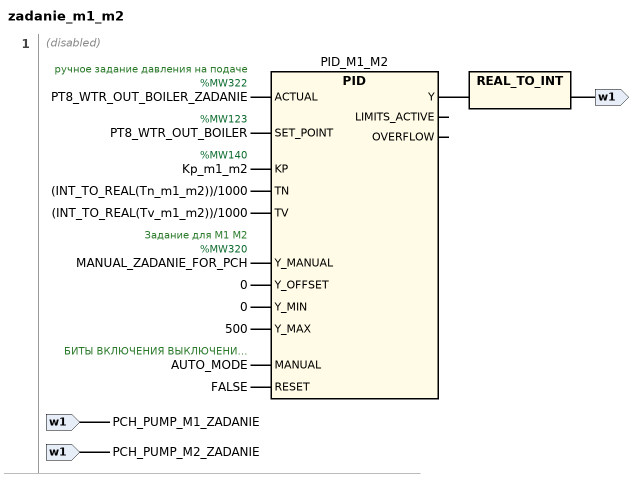
// NETWORK 1 (disabled)
//   PT8_WTR_OUT_BOILER_ZADANIE: ручное задание давления на подаче | AT %MW322
//   PT8_WTR_OUT_BOILER: AT %MW123
//   Kp_m1_m2: AT %MW140
//   MANUAL_ZADANIE_FOR_PCH: Задание для М1 М2 | AT %MW320
//   AUTO_MODE: БИТЫ ВКЛЮЧЕНИЯ ВЫКЛЮЧЕНИЯ МЕХАНИЗМОВ ========== КОНЕЦ ======
// PID_M1_M2(
//     ACTUAL := PT8_WTR_OUT_BOILER_ZADANIE,
//     SET_POINT := PT8_WTR_OUT_BOILER,
//     KP := Kp_m1_m2,
//     TN := (INT_TO_REAL(Tn_m1_m2))/1000,
//     TV := (INT_TO_REAL(Tv_m1_m2))/1000,
//     Y_MANUAL := MANUAL_ZADANIE_FOR_PCH,
//     Y_OFFSET := 0,
//     Y_MIN := 0,
//     Y_MAX := 500,
//     MANUAL := AUTO_MODE,
//     RESET := FALSE); // PID
// _w1 := REAL_TO_INT(PID_M1_M2.Y);
// PCH_PUMP_M1_ZADANIE := _w1;
// PCH_PUMP_M2_ZADANIE := _w1;

END_PROGRAM

// A_TESTS/get_data_from_oven
PROGRAM get_data_from_oven
VAR
	good: BOOL;
END_VAR

(*
IF (step=1) THEN
//ЗАПРОС ОВЕНУ ПОЛУЧИТЬ СОСТОЯНИЕ ВХОДА 1	
	data_to_send[0]:=16#04;//adr
	data_to_send[1]:=16#03;//команда
	data_to_send[2]:=16#00;//старший байт читаемого регистра
	data_to_send[3]:=16#01;//младший байт читаемого регистра
	data_to_send[4]:=16#00;//старший байт количества читаемых регистров
	data_to_send[5]:=16#01;//младший байт количества читаемых регистров
	data_to_send[6]:=16#D5;//CRC
	data_to_send[7]:=16#9F;//CRC 
	

	good := send_to_oven();
	
	IF(good) THEN
		POSITION_VALVE_PEREPUSK:=resv_data_from_ckm[3];
  		POSITION_VALVE_PEREPUSK:=SHL (POSITION_VALVE_PEREPUSK, 8)+resv_data_from_ckm[4];//3 И 4 BYTE В ОТВЕТЕ ЭТО ДАННЫЕ СО ВХОДА 1
	END_IF 		
END_IF


IF(step=2) THEN
//ЗАПРОС ОВЕНУ ПОЛУЧИТЬ СОСТОЯНИЕ ВХОДА 2	
	data_to_send[0]:=16#04;
	data_to_send[1]:=16#03;
	data_to_send[2]:=16#00;
	data_to_send[3]:=16#07;
	data_to_send[4]:=16#00;
	data_to_send[5]:=16#01;
	data_to_send[6]:=16#35;
	data_to_send[7]:=16#9E; 

	good := send();
	
	IF(good) THEN 
  		POSITION_VALVE_HEATER:=resv_data[3];
  		POSITION_VALVE_HEATER:=SHL (POSITION_VALVE_HEATER, 8)+resv_data[4];//3 И 4 BYTE В ОТВЕТЕ ЭТО ДАННЫЕ СО ВХОДА 1	
	END_IF
END_IF
*)

END_PROGRAM
